# EPICS substitutions: testDevApp/Db/user.substitutions
# Example substitutions file

file "db/dbExample1.db" {
    { user = "lucas" }
}

file db/dbExample2.db {
    pattern { user, no, scan }
        { "lucas", 1, "1 second" }
        { "lucas", 2, "2 second" }
        { "lucas", 3, "5 second" }
}
